FUNCTION_BLOCK Pid_Tests EXTENDS FB_TestSuite
VAR
    delta : LREAL := 1E-5;
END_VAR

OnlyProportionalPart();
OnlyPropotionalPartRunTwiceWithDifferentInputs();
OnlyIntegralPart();
OnlyIntegralPartSetPreviousIntegralPartBefore();
OnlyDifferentialPart();
OnlyDifferentialPartWithDiffLimit();

METHOD OnlyDifferentialPart
VAR_INST
    P : Pid;
    parameters : PidParameters := (Kd:=0.01);
END_VAR
TcUnit.TEST('OnlyDifferentialPart');

P(setpoint:=10, actual:=6, parameters:=parameters);
AssertEquals_LREAL(
    Expected:=0.04,
    Actual:=P.Out,
    Delta:=delta,
    Message:='Pid output run 1 not correct'
);

P(setpoint:=10, actual:=8, parameters:=parameters);
AssertEquals_LREAL(
    Expected:=-0.02,
    Actual:=P.Out,
    Delta:=delta,
    Message:='Pid output run 2 not correct'
);

TcUnit.TEST_FINISHED();
END_METHOD

METHOD OnlyDifferentialPartWithDiffLimit
VAR_INST
    P : Pid;
    parameters : PidParameters := (Kd:=0.01);
END_VAR
TcUnit.TEST('OnlyDifferentialPartWithDiffLimit');

P.DifferentialPartLimit := 3;
P(setpoint:=10, actual:=6, parameters:=parameters);
AssertEquals_LREAL(
    Expected:=0,
    Actual:=P.Out,
    Delta:=delta,
    Message:='Pid output run 1 not correct'
);

P(setpoint:=10, actual:=8, parameters:=parameters);
AssertEquals_LREAL(
    Expected:=-0.02,
    Actual:=P.Out,
    Delta:=delta,
    Message:='Pid output run 2 not correct'
);

TcUnit.TEST_FINISHED();
END_METHOD

METHOD OnlyIntegralPart
VAR_INST
    P : Pid;
    parameters : PidParameters := (Ki:=0.25);
END_VAR
TcUnit.TEST('OnlyIntegralPart');

P(setpoint:=10, actual:=6, parameters:=parameters);
AssertEquals_LREAL(
    Expected:=1,
    Actual:=P.Out,
    Delta:=delta,
    Message:='Pid output run 1 not correct'
);

P(setpoint:=10, actual:=8, parameters:=parameters);
AssertEquals_LREAL(
    Expected:=1.5,
    Actual:=P.Out,
    Delta:=delta,
    Message:='Pid output run 2 not correct'
);

TcUnit.TEST_FINISHED();
END_METHOD

METHOD OnlyIntegralPartSetPreviousIntegralPartBefore
VAR_INST
    P : Pid;
    parameters : PidParameters := (Ki:=0.25);
END_VAR
TcUnit.TEST('OnlyIntegralPartSetPreviousIntegralPartBefore');

P.PreviousIntegralPart := 3;

P(setpoint:=10, actual:=6, parameters:=parameters);
AssertEquals_LREAL(
    Expected:=4,
    Actual:=P.Out,
    Delta:=delta,
    Message:='Pid output run 1 not correct'
);

P(setpoint:=10, actual:=8, parameters:=parameters);
AssertEquals_LREAL(
    Expected:=4.5,
    Actual:=P.Out,
    Delta:=delta,
    Message:='Pid output run 2 not correct'
);

TcUnit.TEST_FINISHED();
END_METHOD

METHOD OnlyProportionalPart
VAR_INST
    P : Pid;
    parameters : PidParameters := (Kp:=5);
END_VAR
TcUnit.TEST('OnlyProportionalPart');

P(setpoint:=10, actual:=5, parameters:=parameters);

AssertEquals_LREAL(Expected:=25, Actual:=P.Out, Delta:=delta, Message:='Pid output not correct');

TcUnit.TEST_FINISHED();
END_METHOD

METHOD OnlyPropotionalPartRunTwiceWithDifferentInputs
VAR_INST
    P : Pid;
    parameters : PidParameters := (Kp:=2);
END_VAR
TcUnit.TEST('OnlyPropotionalPartRunTwiceWithDifferentInputs');

P(setpoint:=3, actual:=4.5, parameters:=parameters);

AssertEquals_LREAL(
    Expected:=-3,
    Actual:=P.Out,
    Delta:=delta,
    Message:='Pid output after run 1 not correct'
);

P(setpoint:=-8, actual:=-6, parameters:=parameters);

AssertEquals_LREAL(
    Expected:=-4,
    Actual:=P.Out,
    Delta:=delta,
    Message:='Pid output after run 2 not correct'
);

TcUnit.TEST_FINISHED();
END_METHOD

END_FUNCTION_BLOCK

(* stored: Version 1.1.0.1, ProductVersion 3.1.4024.11
   POU Pid_Tests: Id {d37e3a2d-290f-492c-9ef6-af8dd98f69e3}, SpecialFunc None
   Method OnlyDifferentialPart: Id {4f99075d-a13f-4f18-8a15-c8ddba8e5a52}
   Method OnlyDifferentialPartWithDiffLimit: Id {241d286d-fea2-4eb4-8a87-6d9bdc37a17d}
   Method OnlyIntegralPart: Id {5d97b5ea-7ca7-495f-b7ce-68e585bdb9a4}
   Method OnlyIntegralPartSetPreviousIntegralPartBefore: Id {e14023e9-bbe5-4ab4-b516-86db5b89a50c}
   Method OnlyProportionalPart: Id {4180392b-050f-4fed-a265-d9a44e45b893}
   Method OnlyPropotionalPartRunTwiceWithDifferentInputs: Id {1d265881-ea1f-4b87-98ee-c292edfec96c} *)
